// TIA Portal project "blink" (V16)

(* hardware
DEVICE "S7-1200 station_1"  S7-1200 Station
   slot 0: "Rack_0"  S7-1200 Rack  Rack  V1.0
   slot 1: "PLC_1"  CPU 1212C DC/DC/DC  6ES7 212-1AE40-0XB0  V4.4
*)

// ===== PLC "PLC_1"  CPU 1212C DC/DC/DC =====

VAR_GLOBAL   // PLC tag table "Default tag table"
   "System_Byte" AT %MB1 : Byte;
   "FirstScan" AT %M1.0 : Bool;
   "DiagStatusUpdate" AT %M1.1 : Bool;
   "AlwaysTRUE" AT %M1.2 : Bool;
   "AlwaysFALSE" AT %M1.3 : Bool;
   "Clock_Byte" AT %MB10 : Byte;
   "Clock_10Hz" AT %M10.0 : Bool;
   "Clock_5Hz" AT %M10.1 : Bool;
   "Clock_2.5Hz" AT %M10.2 : Bool;
   "Clock_2Hz" AT %M10.3 : Bool;
   "Clock_1.25Hz" AT %M10.4 : Bool;
   "Clock_1Hz" AT %M10.5 : Bool;
   "Clock_0.625Hz" AT %M10.6 : Bool;
   "Clock_0.5Hz" AT %M10.7 : Bool;
   "Tag_1" AT %Q0.4 : Bool;
   "input" AT %I0.0 : Bool;
   "Tag_4" AT %Q0.2 : Bool;
   "Tag_5" AT %Q0.1 : Bool;
   "Tag_2" AT %M0.0 : Bool;
   "Tag_3" AT %M0.1 : Bool;
   "Tag_6" AT %Q0.0 : Bool;
END_VAR

ORGANIZATION_BLOCK "Main"   // OB1, LAD, ProgramCycle
TITLE = "Main Program Sweep (Cycle)"
{ S7_Optimized_Access := 'TRUE' }
VERSION : 0.1
   VAR_INPUT
      Initial_Call : Bool;   // Initial call of this OB
      Remanence : Bool;   // =True, if remanent data are available
   END_VAR
   VAR_TEMP   // added for the SCL form of the ladder/FBD networks
      _w1 : Bool;
   END_VAR
BEGIN

REGION Network 1
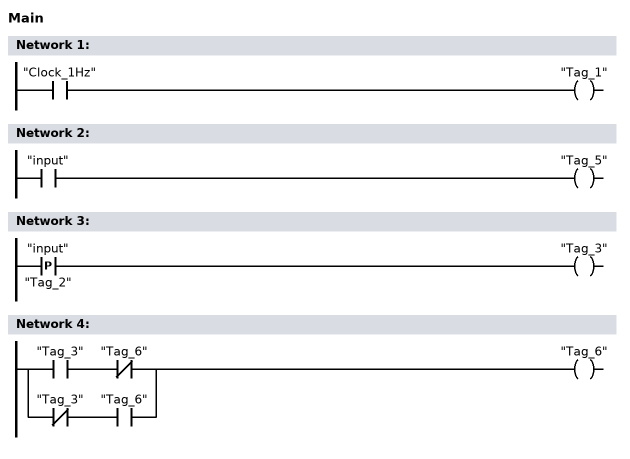
   RUNG wire#powerrail
      Contact( "Clock_1Hz" )
      Coil( "Tag_1" )
   END_RUNG
   // the same network as SCL:
   "Tag_1" := "Clock_1Hz";
END_REGION

REGION Network 2
   RUNG wire#powerrail
      Contact( "input" )
      Coil( "Tag_5" )
   END_RUNG
   // the same network as SCL:
   "Tag_5" := "input";
END_REGION

REGION Network 3
   RUNG wire#powerrail
      P_Contact(operand := "input", bit := "Tag_2")
      Coil( "Tag_3" )
   END_RUNG
   // the same network as SCL:
   #_w1 := "input" AND NOT "Tag_2";   // rising edge of "input"
   "Tag_2" := "input";
   "Tag_3" := #_w1;
END_REGION

REGION Network 4
   RUNG wire#powerrail
      Contact( "Tag_3" )
      I_Contact( "Tag_6" )
      wire#w1
      Coil( "Tag_6" )
   END_RUNG
   RUNG wire#powerrail
      I_Contact( "Tag_3" )
      Contact( "Tag_6" )
   END_RUNG wire#w1
   // the same network as SCL:
   "Tag_6" := ("Tag_3" AND NOT "Tag_6") OR (NOT "Tag_3" AND "Tag_6");
END_REGION
END_ORGANIZATION_BLOCK